{attribute 'qualified_only'}
VAR_GLOBAL
	g_unCleanroomConnect		: UN_CleanroomConnect;
	
	g_eStaLedColor 				: E_KmweLedColors := E_KmweLedColors.Idle;
	g_bLedFlashSlow 			: BOOL;
	g_bLedFlashFast				: BOOL;

	g_fbHmiBtnSimulation		: FB_HmiBtn;
	
	g_sUser						: STRING;
	g_sSerialNumber				: STRING;
	g_sNotesEntry				: T_MAXSTRING;
	
	//Hmi linked variable
	g_sToHmiTopContent			: STRING;
	g_sToHmiMiddleContent		: STRING;
	g_sToHmiBottomContent		: STRING;
	
	//Structs with screens that can be appointed to linked variables
	g_stHmiTopBar				: ST_HmiTopBar;
	g_stHmiMiddle				: ST_HmiMiddle;
	g_stHmiBottomBar			: ST_HmiBottomBar;
	
	g_osrNotify					: R_TRIG;	
END_VAR

VAR_GLOBAL CONSTANT
	g_MAX_LEN_INTERLOCK_REASON : USINT := 64;
	g_LEN_INTERLOCK_LIST : USINT := 6;
END_VAR

(* stored: Version 1.1.0.1, ProductVersion 3.1.4024.12
   GVL GVL: Id {9d829feb-50db-4587-bef7-e7e48dffe79b} *)
